(* IEC 61131-3 sources: Industry-PLC-LLM/data/PLCBEAD_repo/PLCBEAD_PLCEmbed-main/PLC-BEAD/Source/GEB/JD2000, 1 file *)

(* ---- JD2000.ST ---- *)
FUNCTION JD2000:REAL

	VAR_INPUT
		DTI :	UDINT;
	END_VAR

	JD2000 := UDINT_TO_REAL(DTI - UDINT#946728000) / 86400.0;

END_FUNCTION

PROGRAM program0
	VAR
		DTI :	UDINT;
		OUT : REAL;
	END_VAR

	OUT := JD2000(DTI);
END_PROGRAM
